Universal Robots URScript: turntable.script

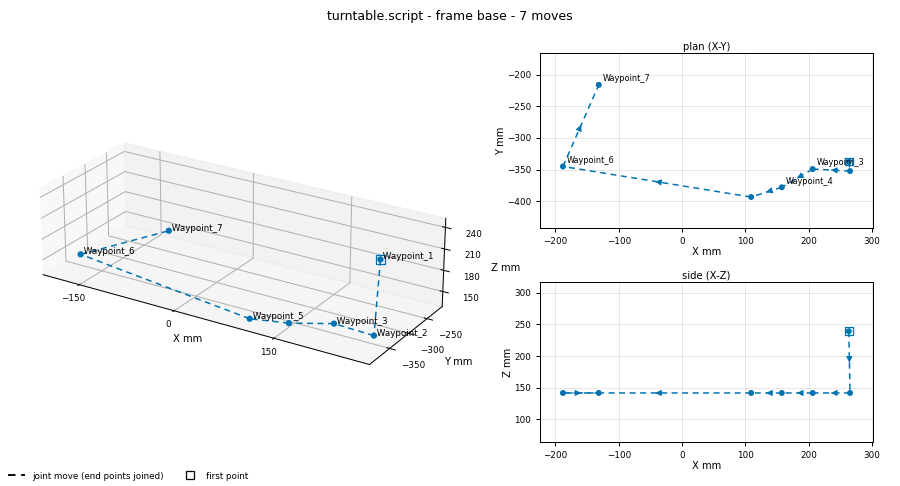
[picture p0: tool path of turntable.script in frame base, 7 of 7 moves have a stored position in this frame; points joined in program order, loops and branches not executed]
def turntable():
  global _hidden_verificationVariable=0
  set_tool_communication(False, 115200, 0, 1, 1.5, 3.5)
  set_tool_output_mode(0)
  set_tool_digital_output_mode(0, 1)
  set_tool_digital_output_mode(1, 1)
  set_tool_voltage(0)
  set_safety_mode_transition_hardness(1)
  set_standard_analog_input_domain(0, 1)
  set_standard_analog_input_domain(1, 1)
  set_tool_analog_input_domain(0, 1)
  set_tool_analog_input_domain(1, 1)
  set_analog_outputdomain(0, 0)
  set_analog_outputdomain(1, 0)
  set_input_actions_to_default()
  set_target_payload(0.530000, [0.009000, -0.039000, 0.092000], [0.000534, 0.000534, 0.000534, 0.000000, 0.000000, 0.000000])
  set_tcp(p[0.0,0.0,0.11,0.0,0.0,0.0])
  set_gravity([0.0, 0.0, 9.82])
  global Al_plate=p[0.12405209206180495,-0.2666666051843552,0.020008101224669964,-9.276623980477388E-5,1.8107917580596192E-5,3.1233857134705927]
  global Frame2x2=p[0.18266245434305164,-0.34273121659514855,0.026002571110600767,-2.225423529876215E-4,3.0110667546023537E-4,3.1233976058306383]
  global URlogoTutorial=p[-0.08178353973148575,-0.3363174165299142,0.04788621506469384,-3.9746155723688456E-5,-3.4682148779121894E-5,-1.5668291789091222]
  global carouselrod=p[0.2020731702281844,-0.34951442511341274,0.1947611446273096,3.139766958234101,-0.10689428010274801,-1.1796370330365635E-5]
  global paper=p[-0.09670794781244417,-0.3283412964648025,0.027665994240809913,-3.2057893450593004E-5,2.867088716161181E-5,-1.6085327915291054]
  global rod=p[0.13368013097420872,-0.41123185103490206,0.09926814901395645,2.2214229924093103,-2.2214158162465862,-2.9165882738638143E-5]
  # begin: URCap Installation Node
  #   Source: External Control, 1.0.5, FZI Research Center for Information Technology
  #   Type: External Control
  # end: URCap Installation Node
  step_count_c0b60bdf_8f3b_4db0_b670_6f220ad7429b = 0.0
  thread Step_Counter_Thread_9e4d85a9_1c70_45fe_9fb9_d5c392e96989():
    while (True):
      step_count_c0b60bdf_8f3b_4db0_b670_6f220ad7429b = step_count_c0b60bdf_8f3b_4db0_b670_6f220ad7429b + 1.0
      sync()
    end
  end
  run Step_Counter_Thread_9e4d85a9_1c70_45fe_9fb9_d5c392e96989()
  global Waypoint_1_p=p[.263501689877, -.337317763427, .239349489480, 3.139797243720, -.105347053477, -.000037720516]
  global Waypoint_1_q=[-0.5959728399859827, -2.1057659588255824, -0.6533136367797852, -1.9525557957091273, 1.5718059539794922, 4.181682586669922]
  global Waypoint_2_p=p[.265438435610, -.352444474661, .141740907029, 3.139726376264, -.105360108121, -.000022031768]
  global Waypoint_2_q=[-0.6231134573565882, -2.1016999683775843, -1.126999020576477, -1.4828875821879883, 1.5722739696502686, 4.154912948608398]
  global Waypoint_3_p=p[.206441973084, -.349241721273, .141737893294, 3.139734184252, -.105329347268, -.000022485776]
  global Waypoint_3_q=[-0.7073677221881312, -1.9410401783385218, -1.3681066036224365, -1.4024366003325959, 1.5721865892410278, 4.070710182189941]
  global Waypoint_4_p=p[.157616611756, -.378012026932, .141738203587, 3.139764187573, -.105376653239, -.000076760662]
  global Waypoint_4_q=[-0.8494070211993616, -1.9579774341978968, -1.3439116477966309, -1.409730003481247, 1.5722019672393799, 3.928692579269409]
  global Waypoint_5_p=p[.109134761588, -.393436595889, .141742225598, 3.139732501163, -.105376381431, -.000050533951]
  global Waypoint_5_q=[-0.972816292439596, -1.9523960552611292, -1.3519116640090942, -1.4072665137103577, 1.5721949338912964, 3.805286407470703]
  global Waypoint_6_p=p[-.188131250090, -.345166366147, .141750553976, 3.139727051239, -.105353578209, -.000024875816]
  global Waypoint_6_q=[-1.7293437162982386, -1.8864180050291957, -1.4439769983291626, -1.381135032778122, 1.572224736213684, 3.0487747192382812]
  global Waypoint_7_p=p[-.131564048097, -.216205376465, .141741700579, 3.139714533984, -.105382776464, -.000044168049]
  global Waypoint_7_q=[-1.572542969380514, -1.2417927545360108, -2.0833356380462646, -1.3863917154124756, 1.571577787399292, 3.2058310508728027]
  $ 2 "Robot Program"
  $ 3 "MoveJ"
  $ 4 "Waypoint_1" "breakAfter"
  set_tcp(p[0.0,0.0,0.11,0.0,0.0,0.0])
  movej(get_inverse_kin(pose_trans(carouselrod, pose_trans(p[-.225374943891, -.334963115579, .194760490893, -3.139766958217, .106894280102, .000011796380], Waypoint_1_p)), qnear=Waypoint_1_q), a=1.3962634015954636, v=0.8235987755982988, r=0.02)
  $ 5 "Waypoint_2" "breakAfter"
  set_tcp(p[0.0,0.0,0.11,0.0,0.0,0.0])
  movej(get_inverse_kin(pose_trans(carouselrod, pose_trans(p[-.225374943891, -.334963115579, .194760490893, -3.139766958217, .106894280102, .000011796380], Waypoint_2_p)), qnear=Waypoint_2_q), a=1.3962634015954636, v=0.8235987755982988, r=0.02)
  $ 6 "Waypoint_3" "breakAfter"
  set_tcp(p[0.0,0.0,0.11,0.0,0.0,0.0])
  movej(get_inverse_kin(pose_trans(carouselrod, pose_trans(p[-.225374943891, -.334963115579, .194760490893, -3.139766958217, .106894280102, .000011796380], Waypoint_3_p)), qnear=Waypoint_3_q), a=1.3962634015954636, v=0.8235987755982988, r=0.02)
  $ 7 "Waypoint_4" "breakAfter"
  set_tcp(p[0.0,0.0,0.11,0.0,0.0,0.0])
  movej(get_inverse_kin(pose_trans(carouselrod, pose_trans(p[-.225374943891, -.334963115579, .194760490893, -3.139766958217, .106894280102, .000011796380], Waypoint_4_p)), qnear=Waypoint_4_q), a=1.3962634015954636, v=0.8235987755982988, r=0.02)
  $ 8 "Waypoint_5" "breakAfter"
  set_tcp(p[0.0,0.0,0.11,0.0,0.0,0.0])
  movej(get_inverse_kin(pose_trans(carouselrod, pose_trans(p[-.225374943891, -.334963115579, .194760490893, -3.139766958217, .106894280102, .000011796380], Waypoint_5_p)), qnear=Waypoint_5_q), a=1.3962634015954636, v=0.8235987755982988, r=0.02)
  $ 9 "MoveJ"
  $ 10 "Waypoint_6" "breakAfter"
  movej(get_inverse_kin(pose_trans(carouselrod, pose_trans(p[-.225374943891, -.334963115579, .194760490893, -3.139766958217, .106894280102, .000011796380], Waypoint_6_p)), qnear=Waypoint_6_q), a=1.3962634015954636, v=0.8141592653589793)
  $ 11 "Wait: 0.3"
  sleep(0.3)
  $ 12 "MoveJ"
  $ 13 "Waypoint_7" "breakAfter"
  movej(get_inverse_kin(pose_trans(carouselrod, pose_trans(p[-.225374943891, -.334963115579, .194760490893, -3.139766958217, .106894280102, .000011796380], Waypoint_7_p)), qnear=Waypoint_7_q), a=1.3962634015954636, v=1.0471975511965976, r=0.02)
end
